Staubli VAL3: frame.dtx

num nClockStatus = 835.53
num nFrame = -1
num nKey = -1
num nRefresh = 59941.087
num nTime = 1
num nView
string sEvent = " 0 World"
public string sItems
string sList[11]
  [0] = " 0 World"
  [1] = " 1 frComparateur"
  [2] = " 2 frPiece"
  [3] = " 3 frame3"
  [4] = " 4 frame4"
  [5] = " 5 frame5"
  [6] = " 6 frame6"
  [7] = " 7 frame7"
  [8] = " 8 frame8"
  [9] = " 9 rd"
  [10] = "10 titi"
string sMenu[8]
  [0] = "Teach"
  [1] = "Tool"
  [2] = "Execute"
  [3] = "ALIGN"
  [4] = "Compute"
  [5] = "Mark"
  [6] = "Paste"
  [7] = "Save"
string sMessage
bool bButton[8]
  [0] = true
  [1] = true
  [2] = true
  [3] = true
  [4] = true
  [5] = true
  [6] = true
  [7] = true
bool bLarge
bool bShowStatus
bool bTrigger
frame fSetFrame = {fatherId=world[0]}
pointRx pCheck = {fatherId=world[0]}
pointRx points[3]
  [0] = {fatherId=world[0]}
  [1] = {fatherId=world[0]}
  [2] = {fatherId=world[0]}
mdesc nom_speed = {tmax=100, rmax=100, blend=off}
mdesc nom_speed_2 = {tmax=1, rmax=1, blend=off}
tool tTool = {fatherId=flange[0], ioLink=valve1}
